INTERFACE I_PackML_Control EXTENDS I_InterfaceBase

METHOD ChangeMode
VAR_INPUT
    Mode : E_PMLUnitMode;
END_VAR
END_METHOD

METHOD ChangeState
VAR_INPUT
    State : E_PMLCommand;
END_VAR
END_METHOD

PROPERTY CurrentMode : E_PMLUnitMode
GET
END_GET
END_PROPERTY

PROPERTY CurrentState : E_PMLState
GET
END_GET
END_PROPERTY

PROPERTY ModeCommand : DINT
GET
END_GET
SET
END_SET
END_PROPERTY

PROPERTY StateCommand : E_PMLCommand
GET
END_GET
SET
END_SET
END_PROPERTY

END_INTERFACE

(* stored: Version 1.1.0.1, ProductVersion 3.1.4024.12
   Itf I_PackML_Control: Id {0a595185-78e0-4efa-95fb-0ab72c8c824d}
   Method ChangeMode: Id {9d75ea51-0646-4dd0-9361-bbe77d2278f4}
   Method ChangeState: Id {dd20a8c0-79ed-4758-b35c-6d9386794f60}
   Property CurrentMode: Id {68aa19f0-a027-4849-bb10-f5584ab8d043}
   Get Get: Id {e4c0be11-49fb-4f99-95fb-f87a759ebdeb}
   Property CurrentState: Id {43595dac-7213-416e-a39c-be01c96ab13c}
   Get Get: Id {21f6fac7-5f70-4bd9-8ec4-66822702fbf5}
   Property ModeCommand: Id {11907bf7-f645-420b-85af-3bf0127cd7f1}
   Get Get: Id {6bf91e32-a7d9-4cd4-a79e-7b430d656783}
   Set Set: Id {0cf2eb2e-aedc-4e54-afcc-be209278627f}
   Property StateCommand: Id {1c454ada-e18d-4933-8772-ef90079bfec6}
   Get Get: Id {8999d4e0-c80d-46d0-9f40-de7660a6e38b}
   Set Set: Id {3495e55a-b4ad-4161-a7ba-1793fe13d390} *)
